# EPICS autosave request: mw100App/Db/MW100_main_settings.req
$(P)$(DAU):C001:Label
$(P)$(DAU):C002:Label
$(P)$(DAU):C003:Label
$(P)$(DAU):C004:Label
$(P)$(DAU):C005:Label
$(P)$(DAU):C006:Label
$(P)$(DAU):C007:Label
$(P)$(DAU):C008:Label
$(P)$(DAU):C009:Label
$(P)$(DAU):C010:Label
$(P)$(DAU):C011:Label
$(P)$(DAU):C012:Label
$(P)$(DAU):C013:Label
$(P)$(DAU):C014:Label
$(P)$(DAU):C015:Label
$(P)$(DAU):C016:Label
$(P)$(DAU):C017:Label
$(P)$(DAU):C018:Label
$(P)$(DAU):C019:Label
$(P)$(DAU):C020:Label
$(P)$(DAU):C021:Label
$(P)$(DAU):C022:Label
$(P)$(DAU):C023:Label
$(P)$(DAU):C024:Label
$(P)$(DAU):C025:Label
$(P)$(DAU):C026:Label
$(P)$(DAU):C027:Label
$(P)$(DAU):C028:Label
$(P)$(DAU):C029:Label
$(P)$(DAU):C030:Label
$(P)$(DAU):C031:Label
$(P)$(DAU):C032:Label
$(P)$(DAU):C033:Label
$(P)$(DAU):C034:Label
$(P)$(DAU):C035:Label
$(P)$(DAU):C036:Label
$(P)$(DAU):C037:Label
$(P)$(DAU):C038:Label
$(P)$(DAU):C039:Label
$(P)$(DAU):C040:Label
$(P)$(DAU):C041:Label
$(P)$(DAU):C042:Label
$(P)$(DAU):C043:Label
$(P)$(DAU):C044:Label
$(P)$(DAU):C045:Label
$(P)$(DAU):C046:Label
$(P)$(DAU):C047:Label
$(P)$(DAU):C048:Label
$(P)$(DAU):C049:Label
$(P)$(DAU):C050:Label
$(P)$(DAU):C051:Label
$(P)$(DAU):C052:Label
$(P)$(DAU):C053:Label
$(P)$(DAU):C054:Label
$(P)$(DAU):C055:Label
$(P)$(DAU):C056:Label
$(P)$(DAU):C057:Label
$(P)$(DAU):C058:Label
$(P)$(DAU):C059:Label
$(P)$(DAU):C060:Label

$(P)$(DAU):A001:Label
$(P)$(DAU):A002:Label
$(P)$(DAU):A003:Label
$(P)$(DAU):A004:Label
$(P)$(DAU):A005:Label
$(P)$(DAU):A006:Label
$(P)$(DAU):A007:Label
$(P)$(DAU):A008:Label
$(P)$(DAU):A009:Label
$(P)$(DAU):A010:Label
$(P)$(DAU):A011:Label
$(P)$(DAU):A012:Label
$(P)$(DAU):A013:Label
$(P)$(DAU):A014:Label
$(P)$(DAU):A015:Label
$(P)$(DAU):A016:Label
$(P)$(DAU):A017:Label
$(P)$(DAU):A018:Label
$(P)$(DAU):A019:Label
$(P)$(DAU):A020:Label
$(P)$(DAU):A021:Label
$(P)$(DAU):A022:Label
$(P)$(DAU):A023:Label
$(P)$(DAU):A024:Label
$(P)$(DAU):A025:Label
$(P)$(DAU):A026:Label
$(P)$(DAU):A027:Label
$(P)$(DAU):A028:Label
$(P)$(DAU):A029:Label
$(P)$(DAU):A030:Label
$(P)$(DAU):A031:Label
$(P)$(DAU):A032:Label
$(P)$(DAU):A033:Label
$(P)$(DAU):A034:Label
$(P)$(DAU):A035:Label
$(P)$(DAU):A036:Label
$(P)$(DAU):A037:Label
$(P)$(DAU):A038:Label
$(P)$(DAU):A039:Label
$(P)$(DAU):A040:Label
$(P)$(DAU):A041:Label
$(P)$(DAU):A042:Label
$(P)$(DAU):A043:Label
$(P)$(DAU):A044:Label
$(P)$(DAU):A045:Label
$(P)$(DAU):A046:Label
$(P)$(DAU):A047:Label
$(P)$(DAU):A048:Label
$(P)$(DAU):A049:Label
$(P)$(DAU):A050:Label
$(P)$(DAU):A051:Label
$(P)$(DAU):A052:Label
$(P)$(DAU):A053:Label
$(P)$(DAU):A054:Label
$(P)$(DAU):A055:Label
$(P)$(DAU):A056:Label
$(P)$(DAU):A057:Label
$(P)$(DAU):A058:Label
$(P)$(DAU):A059:Label
$(P)$(DAU):A060:Label

$(P)$(DAU):K001:Label
$(P)$(DAU):K002:Label
$(P)$(DAU):K003:Label
$(P)$(DAU):K004:Label
$(P)$(DAU):K005:Label
$(P)$(DAU):K006:Label
$(P)$(DAU):K007:Label
$(P)$(DAU):K008:Label
$(P)$(DAU):K009:Label
$(P)$(DAU):K010:Label
$(P)$(DAU):K011:Label
$(P)$(DAU):K012:Label
$(P)$(DAU):K013:Label
$(P)$(DAU):K014:Label
$(P)$(DAU):K015:Label
$(P)$(DAU):K016:Label
$(P)$(DAU):K017:Label
$(P)$(DAU):K018:Label
$(P)$(DAU):K019:Label
$(P)$(DAU):K020:Label
$(P)$(DAU):K021:Label
$(P)$(DAU):K022:Label
$(P)$(DAU):K023:Label
$(P)$(DAU):K024:Label
$(P)$(DAU):K025:Label
$(P)$(DAU):K026:Label
$(P)$(DAU):K027:Label
$(P)$(DAU):K028:Label
$(P)$(DAU):K029:Label
$(P)$(DAU):K030:Label
$(P)$(DAU):K031:Label
$(P)$(DAU):K032:Label
$(P)$(DAU):K033:Label
$(P)$(DAU):K034:Label
$(P)$(DAU):K035:Label
$(P)$(DAU):K036:Label
$(P)$(DAU):K037:Label
$(P)$(DAU):K038:Label
$(P)$(DAU):K039:Label
$(P)$(DAU):K040:Label
$(P)$(DAU):K041:Label
$(P)$(DAU):K042:Label
$(P)$(DAU):K043:Label
$(P)$(DAU):K044:Label
$(P)$(DAU):K045:Label
$(P)$(DAU):K046:Label
$(P)$(DAU):K047:Label
$(P)$(DAU):K048:Label
$(P)$(DAU):K049:Label
$(P)$(DAU):K050:Label
$(P)$(DAU):K051:Label
$(P)$(DAU):K052:Label
$(P)$(DAU):K053:Label
$(P)$(DAU):K054:Label
$(P)$(DAU):K055:Label
$(P)$(DAU):K056:Label
$(P)$(DAU):K057:Label
$(P)$(DAU):K058:Label
$(P)$(DAU):K059:Label
$(P)$(DAU):K060:Label
